INTERFACE ITF_HMIConfigure

METHOD PUBLIC AddConfiguration : BOOL
VAR_INPUT
	fbConfigure		: ITF_HMIConfiguration;
END_VAR
END_METHOD

METHOD PUBLIC Configure : BOOL
VAR_INPUT
	fbHMIManager			: ITF_HMIManagerConfigure;
END_VAR
END_METHOD

END_INTERFACE

(* stored: Version 1.1.0.1
   Itf ITF_HMIConfigure: Id {ee035145-d6e4-4092-9d0a-50f12b14f82b}
   Method AddConfiguration: Id {33ffb79c-1b8e-4f62-b6a6-1fa2a7db8629}
   Method Configure: Id {eeb9239e-d327-4e6b-a63b-9dac7e02c31c} *)
